{attribute 'qualified_only'}
{attribute 'strict'}
TYPE Read_State :
(
	Triggerd := 0,
	DataWritten := 1,
	Done := 2
)UINT;
END_TYPE

(* stored: Version 1.1.0.1, ProductVersion 3.1.4024.10
   DUT Read_State: Id {69bb9099-da6d-4868-863f-d1ca42fcf096} *)
